FUNCTION_BLOCK Controller
  (* Standard: 61499-2 *)
  (* Version 0,1, 2015-00-10, Th?o, PC_THEO *)
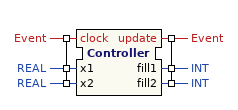
  EVENT_INPUT
    clock WITH x1, x2;
  END_EVENT
  EVENT_OUTPUT
    update WITH fill1, fill2;
  END_EVENT
  VAR_INPUT
    x1 : REAL;
    x2 : REAL;
  END_VAR
  VAR_OUTPUT
    fill1 : INT;
    fill2 : INT;
  END_VAR
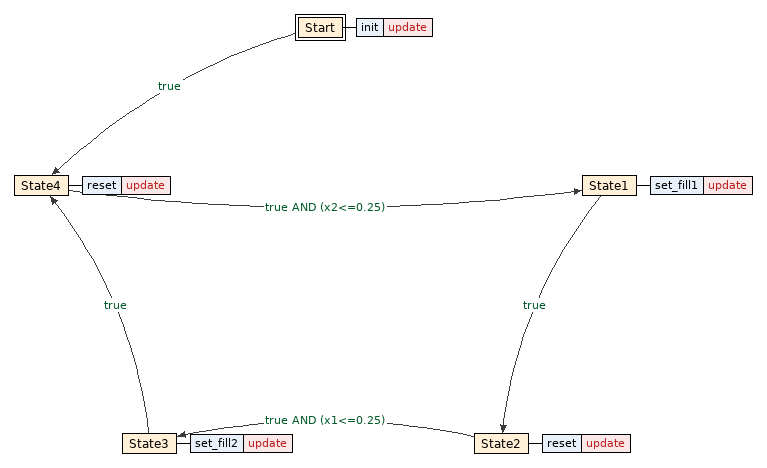
  EC_STATES
    Start : init -> update;
    State1 : set_fill1 -> update;
    State2 : reset -> update;
    State3 : set_fill2 -> update;
    State4 : reset -> update;
  END_STATES
  EC_TRANSITIONS
    Start TO State4 := true;
    State1 TO State2 := true;
    State2 TO State3 := true AND (x1<=0.25);
    State3 TO State4 := true;
    State4 TO State1 := true AND (x2<=0.25);
  END_TRANSITIONS
  ALGORITHM init IN C:
me->fill1=0;me->fill2=0;
me->x1=0.5;me->x2=0.5;
  END_ALGORITHM
  ALGORITHM set_fill1 IN C:
me->fill1=1;
  END_ALGORITHM
  ALGORITHM set_fill2 IN C:
me->fill2=1;
  END_ALGORITHM
  ALGORITHM reset IN C:
me->fill1=0;me->fill2=0;
  END_ALGORITHM
END_FUNCTION_BLOCK
